// TIA Portal V17 export
BLOCK "FC_Unknown"   // ObjectSW21, LAD
BEGIN

REGION Network 1: unknown part
END_REGION
END_BLOCK
